FUNCTION_BLOCK FB_TestBase EXTENDS FB_Base

VAR
END_VAR

END_FUNCTION_BLOCK

(* stored: Version 1.1.0.1
   POU FB_TestBase: Id {e042edc1-8cb1-46b2-9ebe-07265f3d7493}, SpecialFunc None *)
